Staubli VAL3: stringToArray.pgx

public program stringToArray(string x_sString (dimensions=1), string& x_sArray[] (dimensions=1))
// copy one String into an ARRAY of String
  local num i
  local num l_nItem
  local string l_sChar
  local string l_sEmpty
begin
  // define the char use to divide the items
  // PRIORITY
  //  ^
  //  ;
  //  ,
  //
  if find(x_sString,"^")==-1
    if find(x_sString,";")==-1
      l_sChar=","
    else
      l_sChar=";"
    endIf
  else
    l_sChar="^"
  endIf
  // init the X_sArray
  l_sEmpty=""
  call stringCopy(l_sEmpty,x_sArray)
  l_nItem=0
  do
    // increase the ARRAY SIZE
    if l_nItem>0
      insert(x_sArray[l_nItem])
    endIf
    i=find(x_sString,l_sChar)
    // look if was found
    if i!=-1
      // PUT INSIDE THE ARRAY THE STRING
      x_sArray[l_nItem]=left(x_sString,i)
      x_sString=delete(x_sString,i+1,0)
    else
      // look if is empty or not
      if len(x_sString)>0
        x_sArray[l_nItem]=(x_sString)
      endIf
    endIf
    l_nItem=l_nItem+1
  until i==-1
end
